(* Logix 5000 project; controller STAT 1756-L72 rev 20.12; software revision 20.04; part 28 of 34 *)
(* tags used below, declared in another part *)
   B3 : DINT[35];
   N20 : DINT[50];
   N7 : DINT[150];
   N9 : DINT[200];
   T4 : TIMER[100];
   L2_L3_ppas : DINT;
   l2va2 : BOOL;
   l2va3 : BOOL;
   l3va1 : BOOL;
   l3va2 : BOOL;
   l3va3 : BOOL;
   l3va4 : BOOL;
   naohL1VA4 : BOOL;
   naohL2VA4 : BOOL;
   stocklancy3 : DINT;
(* LANCY, continued *)

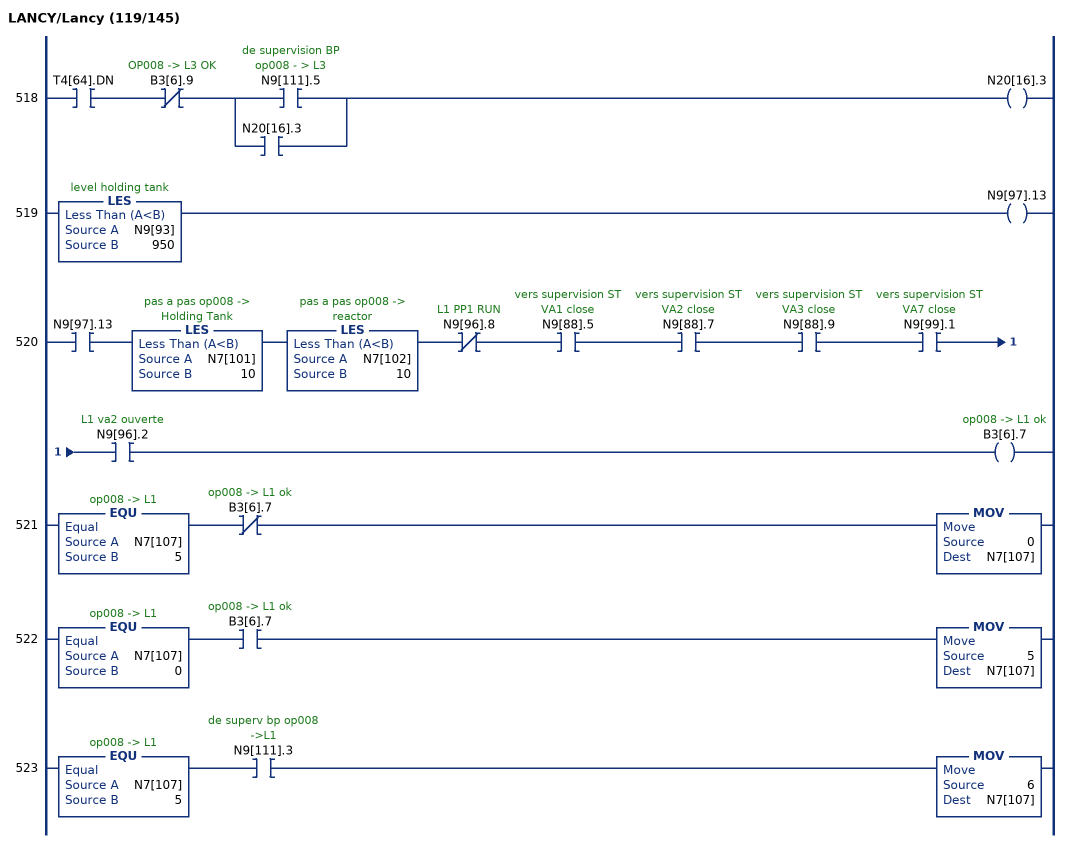
   518: XIC(T4[64].DN)XIO(B3[6].9)[XIC(N9[111].5) ,XIC(N20[16].3) ]OTE(N20[16].3);
   519: LES(N9[93],950)OTE(N9[97].13);
   520: XIC(N9[97].13)LES(N7[101],10)LES(N7[102],10)XIO(N9[96].8)XIC(N9[88].5)XIC(N9[88].7)XIC(N9[88].9)XIC(N9[99].1)XIC(N9[96].2)OTE(B3[6].7);
   521: EQU(N7[107],5)XIO(B3[6].7)MOV(0,N7[107]);
   522: EQU(N7[107],0)XIC(B3[6].7)MOV(5,N7[107]);
   523: EQU(N7[107],5)XIC(N9[111].3)MOV(6,N7[107]);
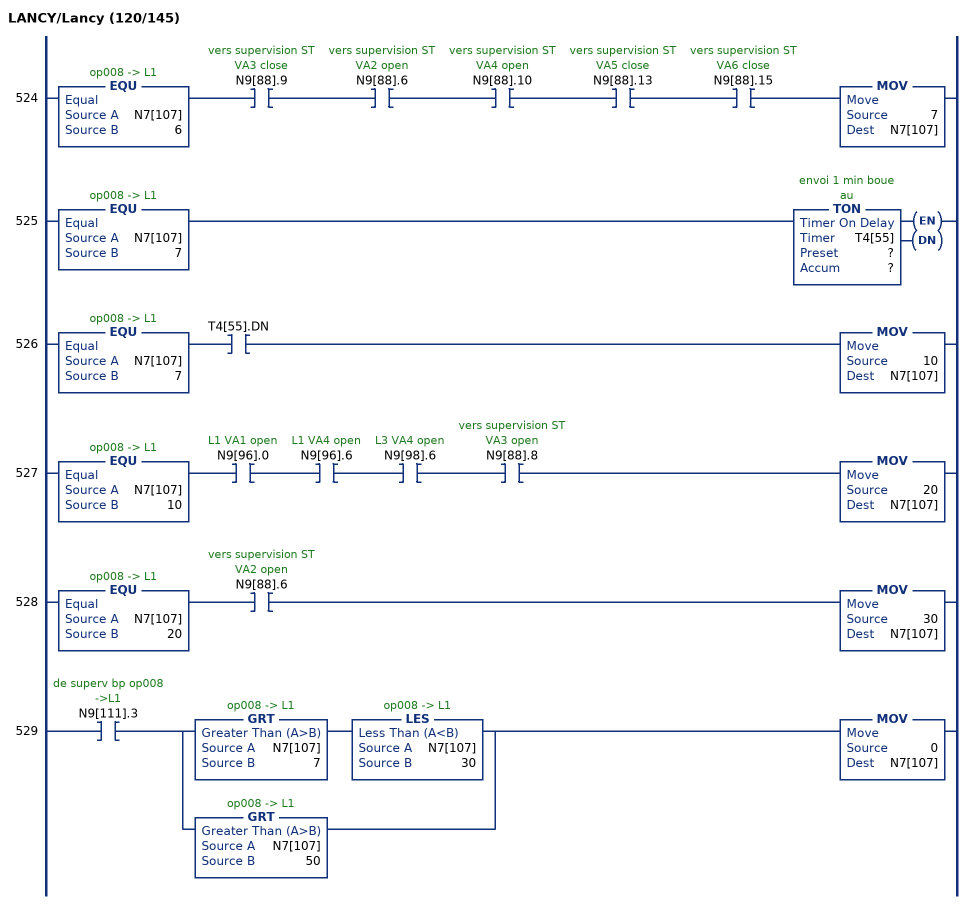
   524: EQU(N7[107],6)XIC(N9[88].9)XIC(N9[88].6)XIC(N9[88].10)XIC(N9[88].13)XIC(N9[88].15)MOV(7,N7[107]);
   525: EQU(N7[107],7)TON(T4[55],?,?);
   526: EQU(N7[107],7)XIC(T4[55].DN)MOV(10,N7[107]);
   527: EQU(N7[107],10)XIC(N9[96].0)XIC(N9[96].6)XIC(N9[98].6)XIC(N9[88].8)MOV(20,N7[107]);
   528: EQU(N7[107],20)XIC(N9[88].6)MOV(30,N7[107]);
   529: XIC(N9[111].3)[GRT(N7[107],7) LES(N7[107],30) ,GRT(N7[107],50) ]MOV(0,N7[107]);
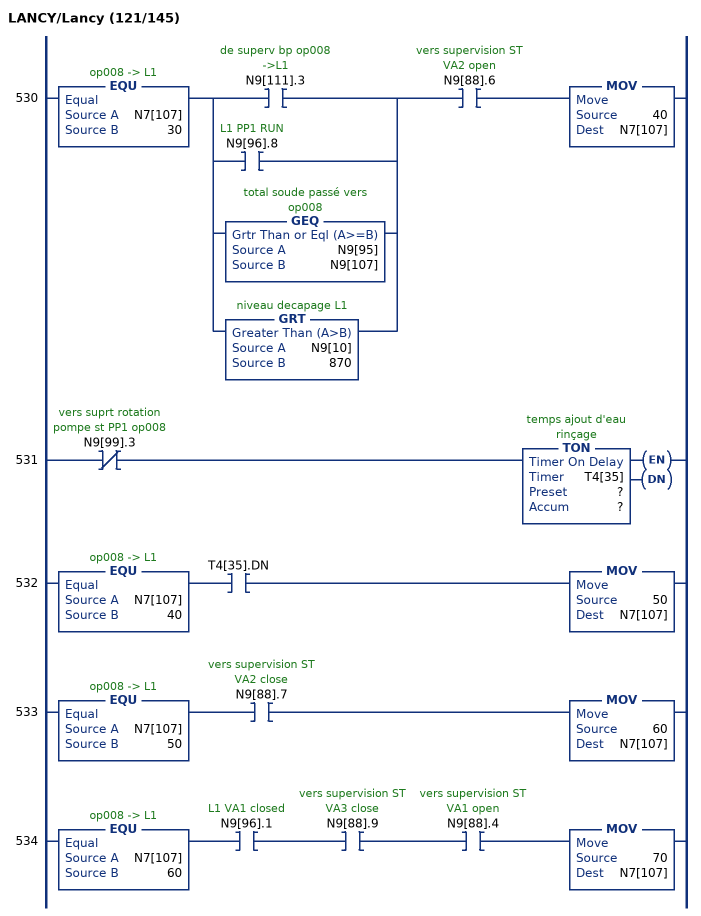
   530: EQU(N7[107],30)[XIC(N9[111].3) ,XIC(N9[96].8) ,GEQ(N9[95],N9[107]) ,GRT(N9[10],870) ]XIC(N9[88].6)MOV(40,N7[107]);
   531: XIO(N9[99].3)TON(T4[35],?,?);
   532: EQU(N7[107],40)XIC(T4[35].DN)MOV(50,N7[107]);
   533: EQU(N7[107],50)XIC(N9[88].7)MOV(60,N7[107]);
   534: EQU(N7[107],60)XIC(N9[96].1)XIC(N9[88].9)XIC(N9[88].4)MOV(70,N7[107]);
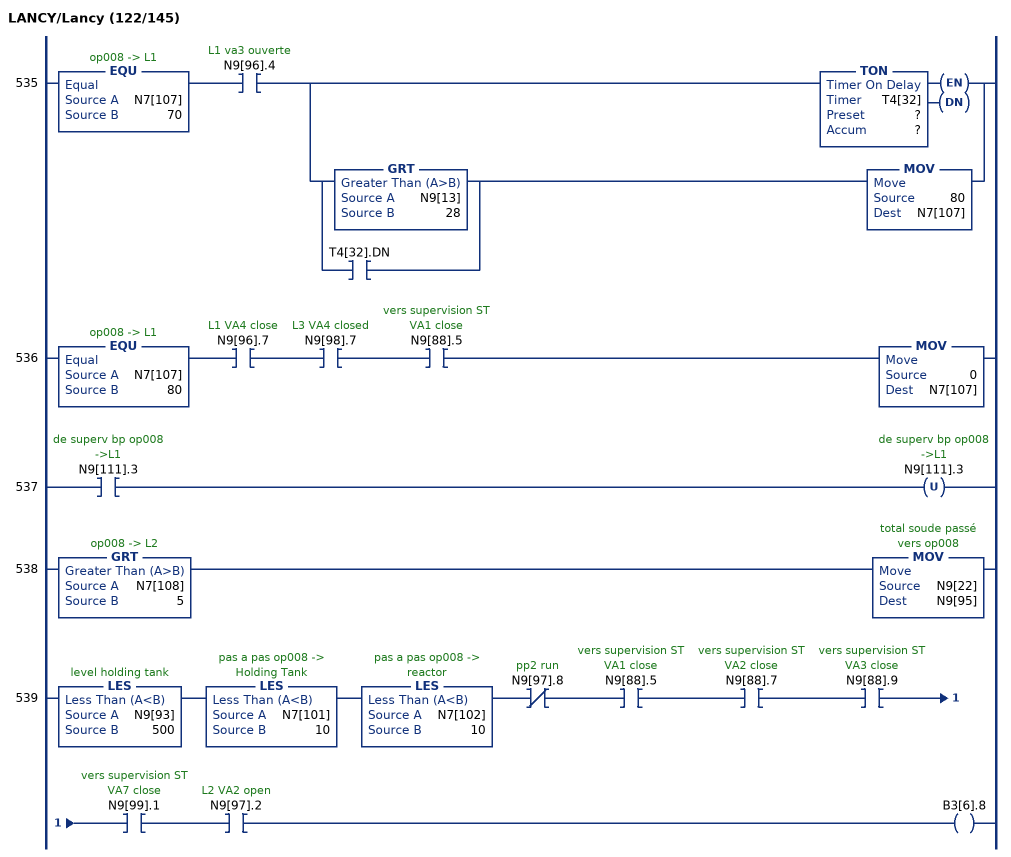
   535: EQU(N7[107],70)XIC(N9[96].4)[TON(T4[32],?,?) ,[GRT(N9[13],28) ,XIC(T4[32].DN) ] MOV(80,N7[107]) ];
   536: EQU(N7[107],80)XIC(N9[96].7)XIC(N9[98].7)XIC(N9[88].5)MOV(0,N7[107]);
   537: XIC(N9[111].3)OTU(N9[111].3);
   538: GRT(N7[108],5)MOV(N9[22],N9[95]);
   539: LES(N9[93],500)LES(N7[101],10)LES(N7[102],10)XIO(N9[97].8)XIC(N9[88].5)XIC(N9[88].7)XIC(N9[88].9)XIC(N9[99].1)XIC(N9[97].2)OTE(B3[6].8);
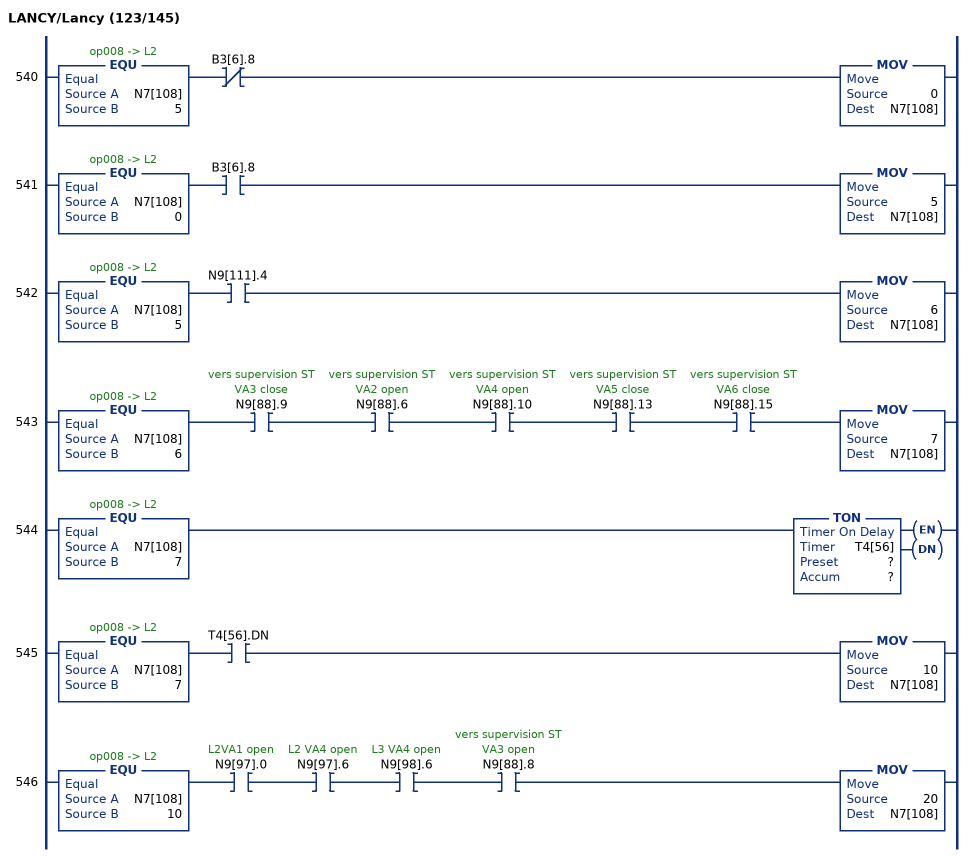
   540: EQU(N7[108],5)XIO(B3[6].8)MOV(0,N7[108]);
   541: EQU(N7[108],0)XIC(B3[6].8)MOV(5,N7[108]);
   542: EQU(N7[108],5)XIC(N9[111].4)MOV(6,N7[108]);
   543: EQU(N7[108],6)XIC(N9[88].9)XIC(N9[88].6)XIC(N9[88].10)XIC(N9[88].13)XIC(N9[88].15)MOV(7,N7[108]);
   544: EQU(N7[108],7)TON(T4[56],?,?);
   545: EQU(N7[108],7)XIC(T4[56].DN)MOV(10,N7[108]);
   546: EQU(N7[108],10)XIC(N9[97].0)XIC(N9[97].6)XIC(N9[98].6)XIC(N9[88].8)MOV(20,N7[108]);
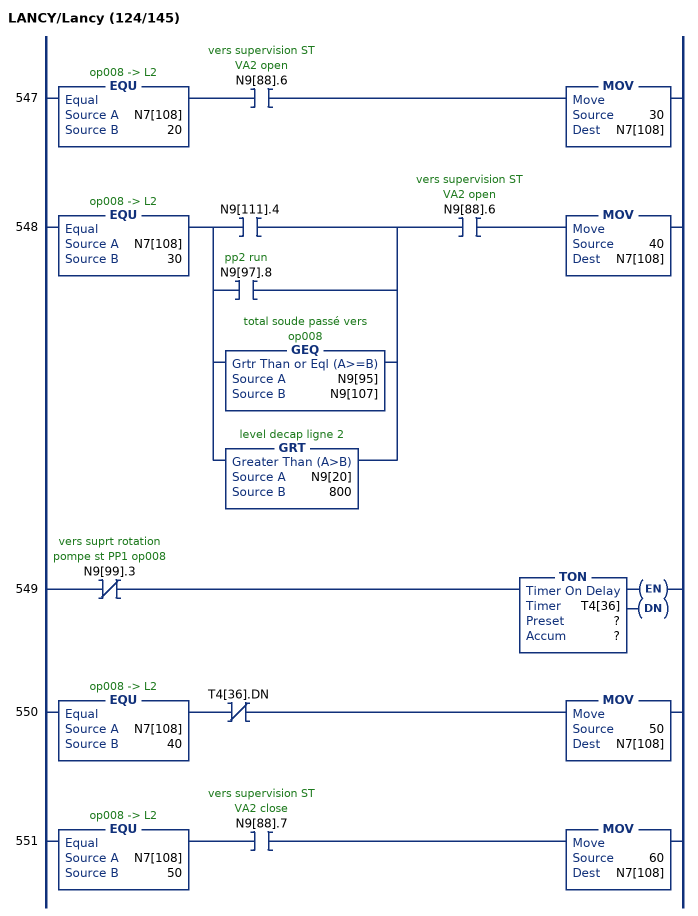
   547: EQU(N7[108],20)XIC(N9[88].6)MOV(30,N7[108]);
   548: EQU(N7[108],30)[XIC(N9[111].4) ,XIC(N9[97].8) ,GEQ(N9[95],N9[107]) ,GRT(N9[20],800) ]XIC(N9[88].6)MOV(40,N7[108]);
   549: XIO(N9[99].3)TON(T4[36],?,?);
   550: EQU(N7[108],40)XIO(T4[36].DN)MOV(50,N7[108]);
   551: EQU(N7[108],50)XIC(N9[88].7)MOV(60,N7[108]);
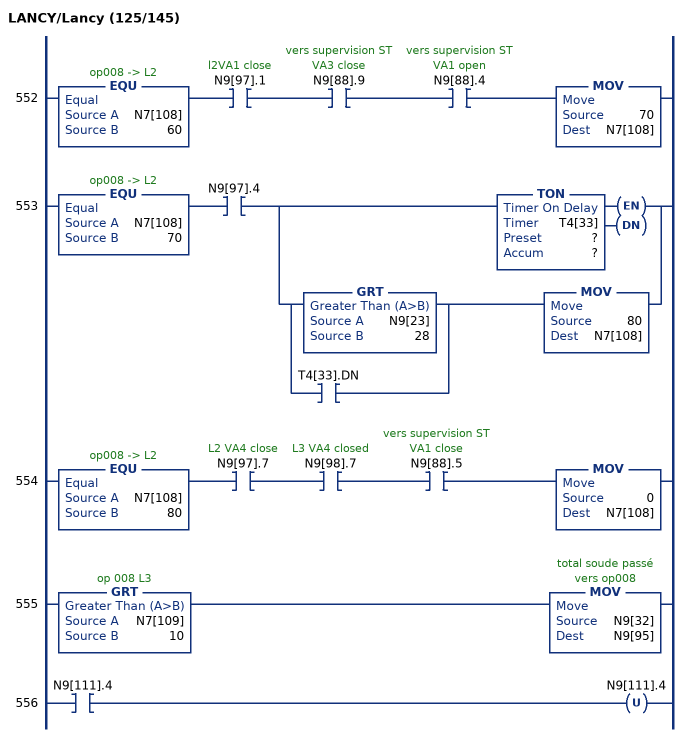
   552: EQU(N7[108],60)XIC(N9[97].1)XIC(N9[88].9)XIC(N9[88].4)MOV(70,N7[108]);
   553: EQU(N7[108],70)XIC(N9[97].4)[TON(T4[33],?,?) ,[GRT(N9[23],28) ,XIC(T4[33].DN) ] MOV(80,N7[108]) ];
   554: EQU(N7[108],80)XIC(N9[97].7)XIC(N9[98].7)XIC(N9[88].5)MOV(0,N7[108]);
   555: GRT(N7[109],10)MOV(N9[32],N9[95]);
   556: XIC(N9[111].4)OTU(N9[111].4);
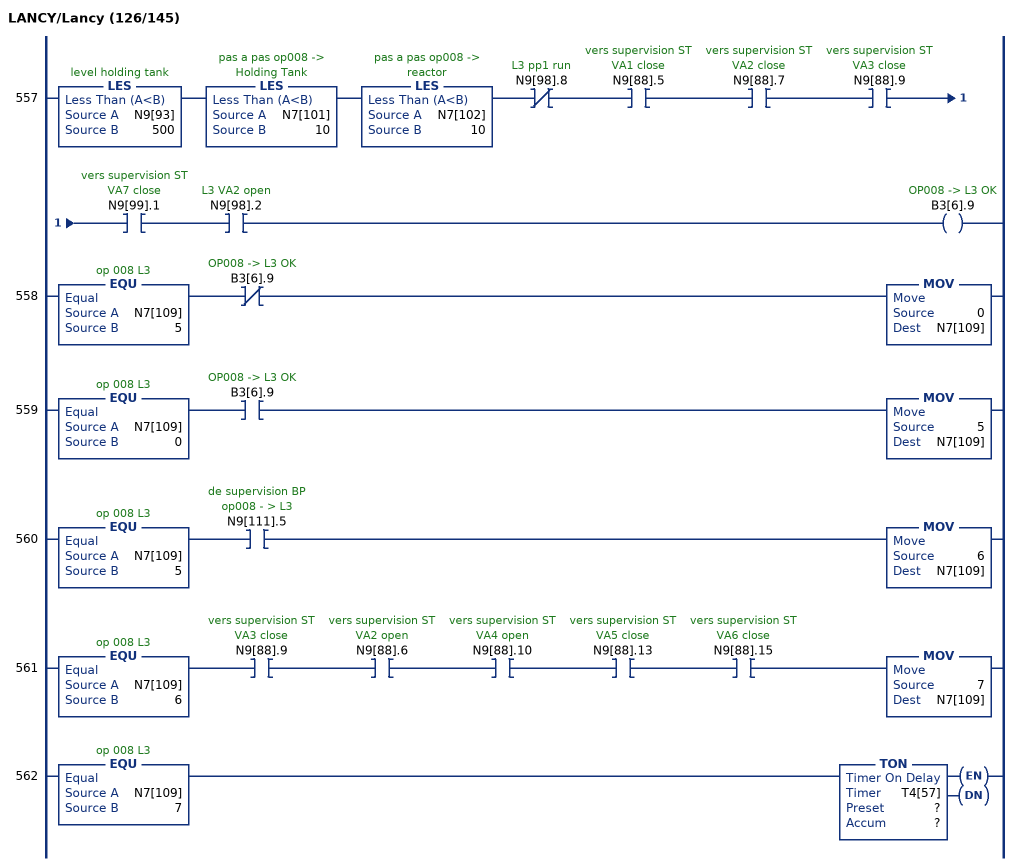
   557: LES(N9[93],500)LES(N7[101],10)LES(N7[102],10)XIO(N9[98].8)XIC(N9[88].5)XIC(N9[88].7)XIC(N9[88].9)XIC(N9[99].1)XIC(N9[98].2)OTE(B3[6].9);
   558: EQU(N7[109],5)XIO(B3[6].9)MOV(0,N7[109]);
   559: EQU(N7[109],0)XIC(B3[6].9)MOV(5,N7[109]);
   560: EQU(N7[109],5)XIC(N9[111].5)MOV(6,N7[109]);
   561: EQU(N7[109],6)XIC(N9[88].9)XIC(N9[88].6)XIC(N9[88].10)XIC(N9[88].13)XIC(N9[88].15)MOV(7,N7[109]);
   562: EQU(N7[109],7)TON(T4[57],?,?);
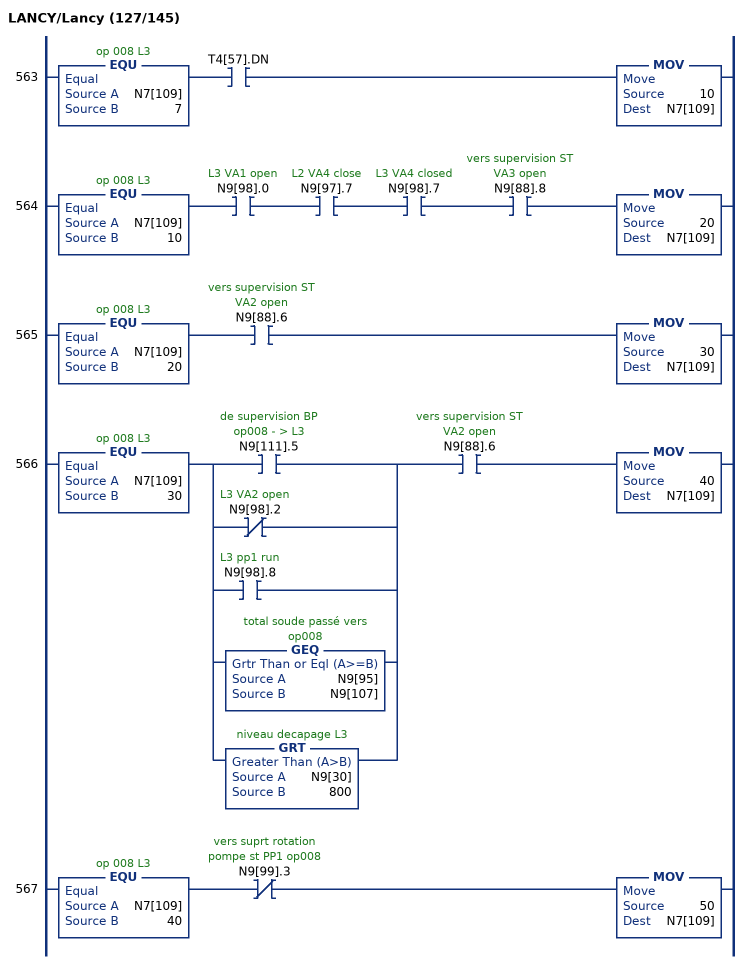
   563: EQU(N7[109],7)XIC(T4[57].DN)MOV(10,N7[109]);
   564: EQU(N7[109],10)XIC(N9[98].0)XIC(N9[97].7)XIC(N9[98].7)XIC(N9[88].8)MOV(20,N7[109]);
   565: EQU(N7[109],20)XIC(N9[88].6)MOV(30,N7[109]);
   566: EQU(N7[109],30)[XIC(N9[111].5) ,XIO(N9[98].2) ,XIC(N9[98].8) ,GEQ(N9[95],N9[107]) ,GRT(N9[30],800) ]XIC(N9[88].6)MOV(40,N7[109]);
   567: EQU(N7[109],40)XIO(N9[99].3)MOV(50,N7[109]);
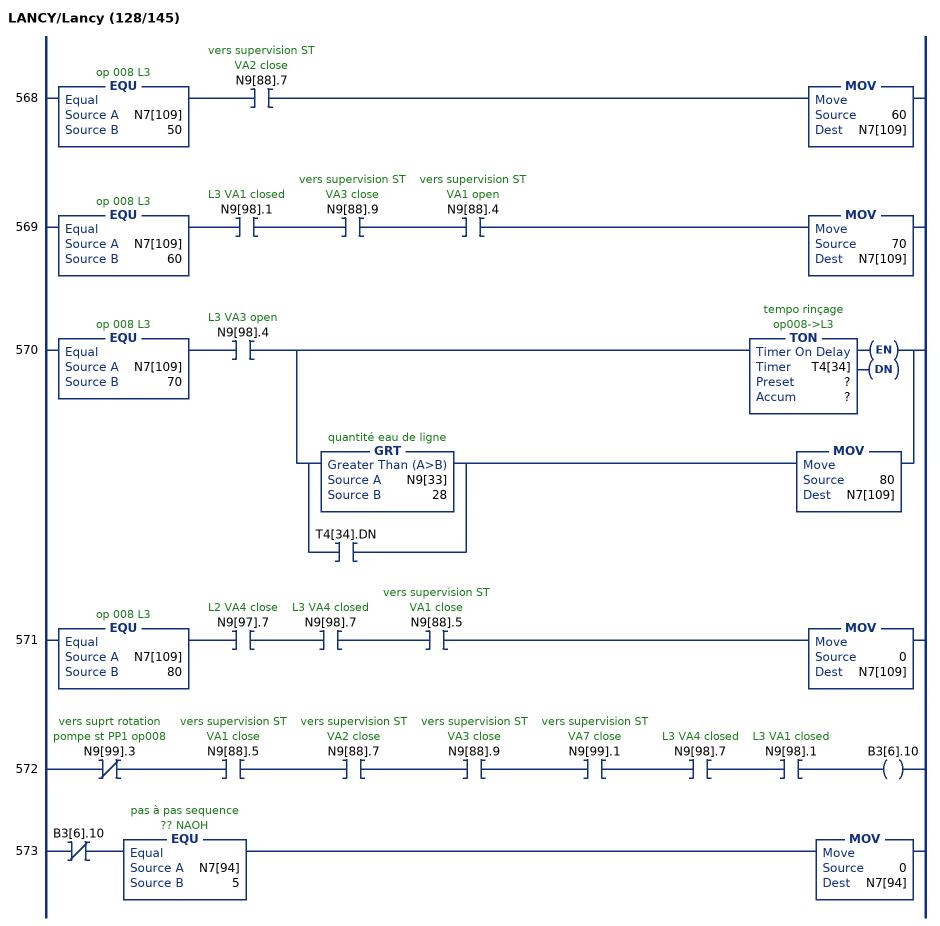
   568: EQU(N7[109],50)XIC(N9[88].7)MOV(60,N7[109]);
   569: EQU(N7[109],60)XIC(N9[98].1)XIC(N9[88].9)XIC(N9[88].4)MOV(70,N7[109]);
   570: EQU(N7[109],70)XIC(N9[98].4)[TON(T4[34],?,?) ,[GRT(N9[33],28) ,XIC(T4[34].DN) ] MOV(80,N7[109]) ];
   571: EQU(N7[109],80)XIC(N9[97].7)XIC(N9[98].7)XIC(N9[88].5)MOV(0,N7[109]);
   572: XIO(N9[99].3)XIC(N9[88].5)XIC(N9[88].7)XIC(N9[88].9)XIC(N9[99].1)XIC(N9[98].7)XIC(N9[98].1)OTE(B3[6].10);
   573: XIO(B3[6].10)EQU(N7[94],5)MOV(0,N7[94]);
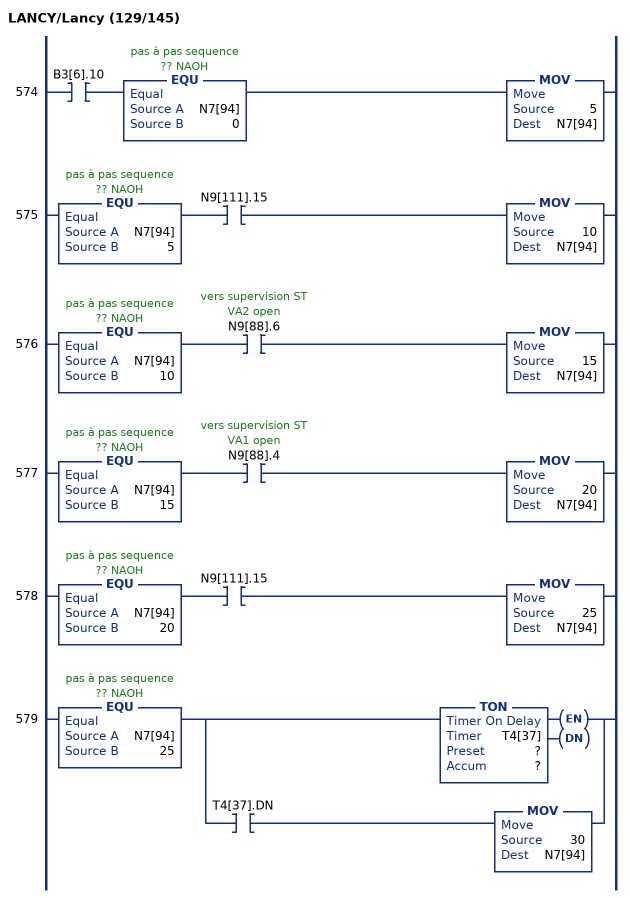
   574: XIC(B3[6].10)EQU(N7[94],0)MOV(5,N7[94]);
   575: EQU(N7[94],5)XIC(N9[111].15)MOV(10,N7[94]);
   576: EQU(N7[94],10)XIC(N9[88].6)MOV(15,N7[94]);
   577: EQU(N7[94],15)XIC(N9[88].4)MOV(20,N7[94]);
   578: EQU(N7[94],20)XIC(N9[111].15)MOV(25,N7[94]);
   579: EQU(N7[94],25)[TON(T4[37],?,?) ,XIC(T4[37].DN) MOV(30,N7[94]) ];
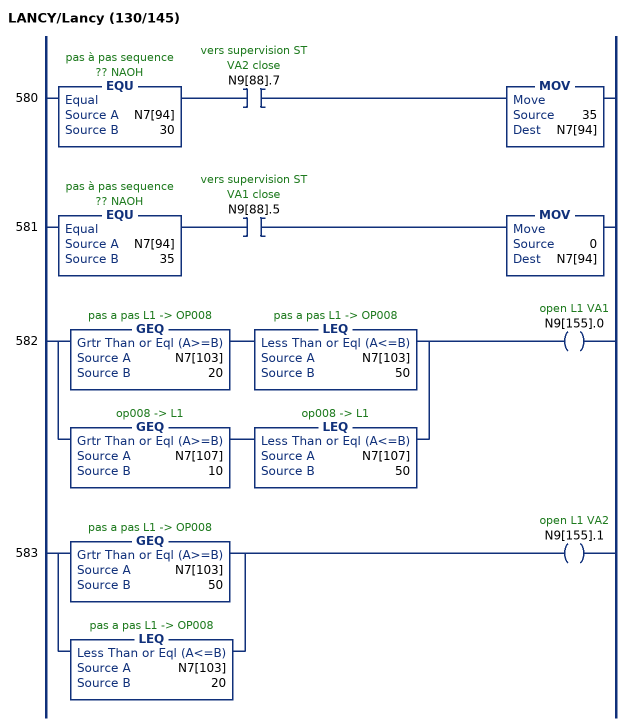
   580: EQU(N7[94],30)XIC(N9[88].7)MOV(35,N7[94]);
   581: EQU(N7[94],35)XIC(N9[88].5)MOV(0,N7[94]);
   582: [GEQ(N7[103],20) LEQ(N7[103],50) ,GEQ(N7[107],10) LEQ(N7[107],50) ]OTE(N9[155].0);
   583: [GEQ(N7[103],50) ,LEQ(N7[103],20) ]OTE(N9[155].1);
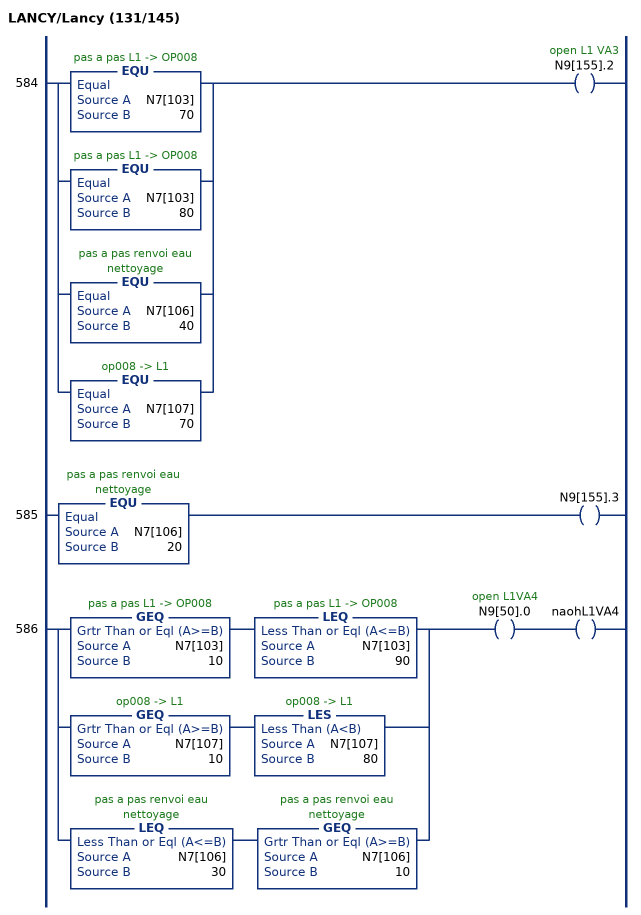
   584: [EQU(N7[103],70) ,EQU(N7[103],80) ,EQU(N7[106],40) ,EQU(N7[107],70) ]OTE(N9[155].2);
   585: EQU(N7[106],20)OTE(N9[155].3);
   586: [GEQ(N7[103],10) LEQ(N7[103],90) ,GEQ(N7[107],10) LES(N7[107],80) ,LEQ(N7[106],30) GEQ(N7[106],10) ]OTE(N9[50].0)OTE(naohL1VA4);
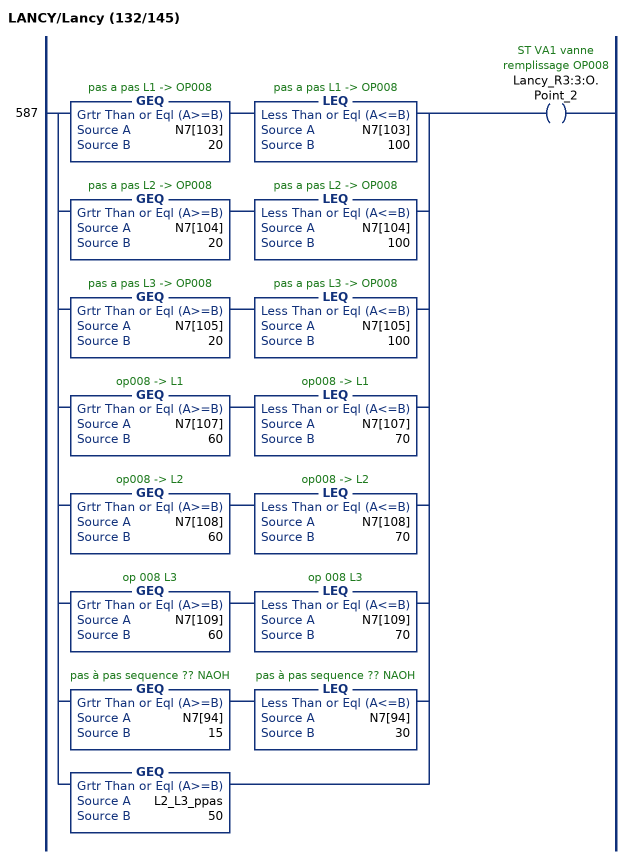
   587: [GEQ(N7[103],20) LEQ(N7[103],100) ,GEQ(N7[104],20) LEQ(N7[104],100) ,GEQ(N7[105],20) LEQ(N7[105],100) ,GEQ(N7[107],60) LEQ(N7[107],70) ,GEQ(N7[108],60) LEQ(N7[108],70) ,GEQ(N7[109],60) LEQ(N7[109],70) ,GEQ(N7[94],15) LEQ(N7[94],30) ,GEQ(L2_L3_ppas,50) ]OTE(Lancy_R3:3:O.Point_2);
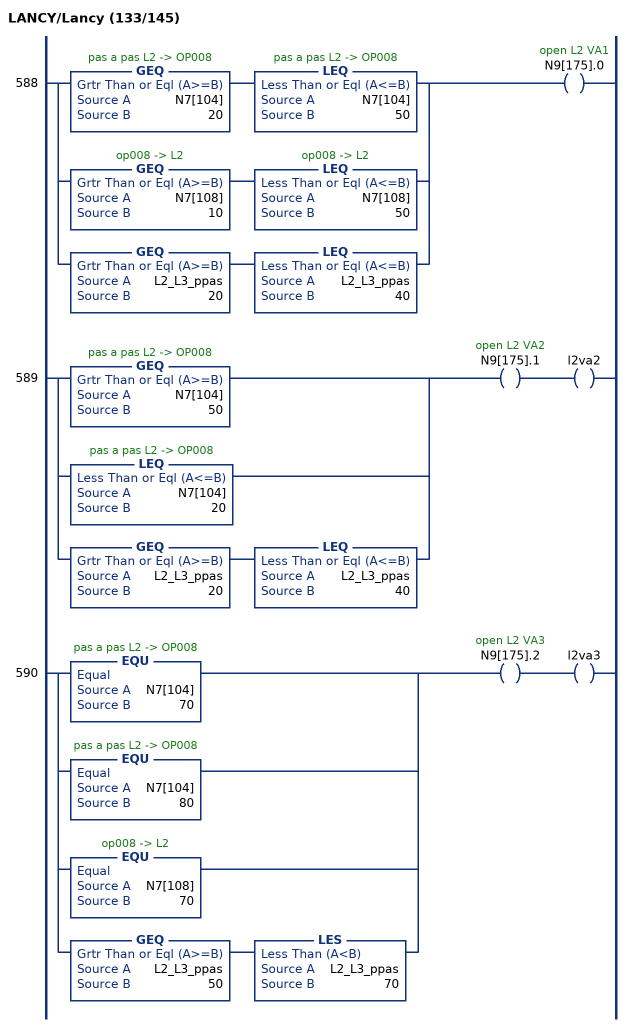
   588: [GEQ(N7[104],20) LEQ(N7[104],50) ,GEQ(N7[108],10) LEQ(N7[108],50) ,GEQ(L2_L3_ppas,20) LEQ(L2_L3_ppas,40) ]OTE(N9[175].0);
   589: [GEQ(N7[104],50) ,LEQ(N7[104],20) ,GEQ(L2_L3_ppas,20) LEQ(L2_L3_ppas,40) ]OTE(N9[175].1)OTE(l2va2);
   590: [EQU(N7[104],70) ,EQU(N7[104],80) ,EQU(N7[108],70) ,GEQ(L2_L3_ppas,50) LES(L2_L3_ppas,70) ]OTE(N9[175].2)OTE(l2va3);
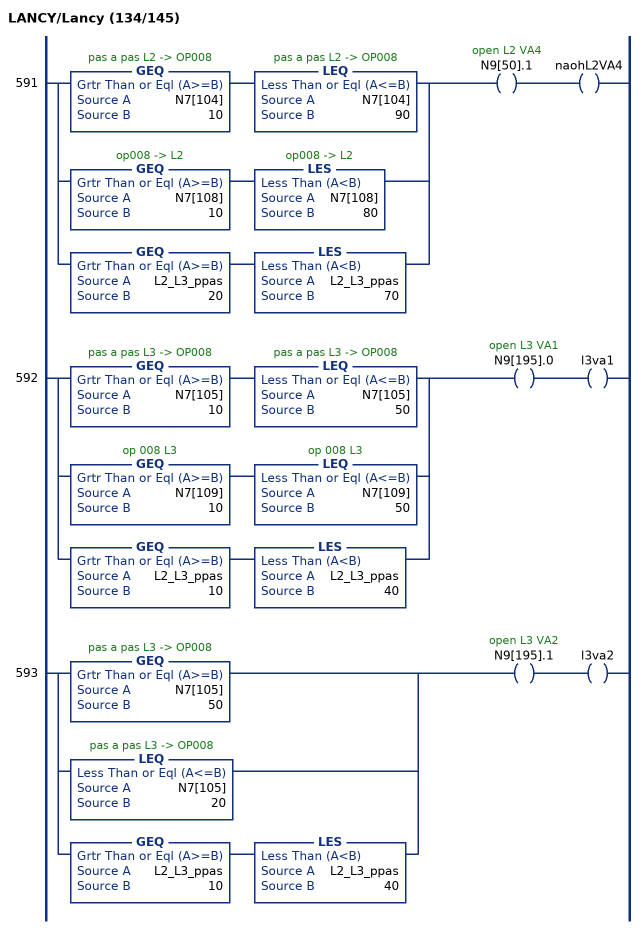
   591: [GEQ(N7[104],10) LEQ(N7[104],90) ,GEQ(N7[108],10) LES(N7[108],80) ,GEQ(L2_L3_ppas,20) LES(L2_L3_ppas,70) ]OTE(N9[50].1)OTE(naohL2VA4);
   592: [GEQ(N7[105],10) LEQ(N7[105],50) ,GEQ(N7[109],10) LEQ(N7[109],50) ,GEQ(L2_L3_ppas,10) LES(L2_L3_ppas,40) ]OTE(N9[195].0)OTE(l3va1);
   593: [GEQ(N7[105],50) ,LEQ(N7[105],20) ,GEQ(L2_L3_ppas,10) LES(L2_L3_ppas,40) ]OTE(N9[195].1)OTE(l3va2);
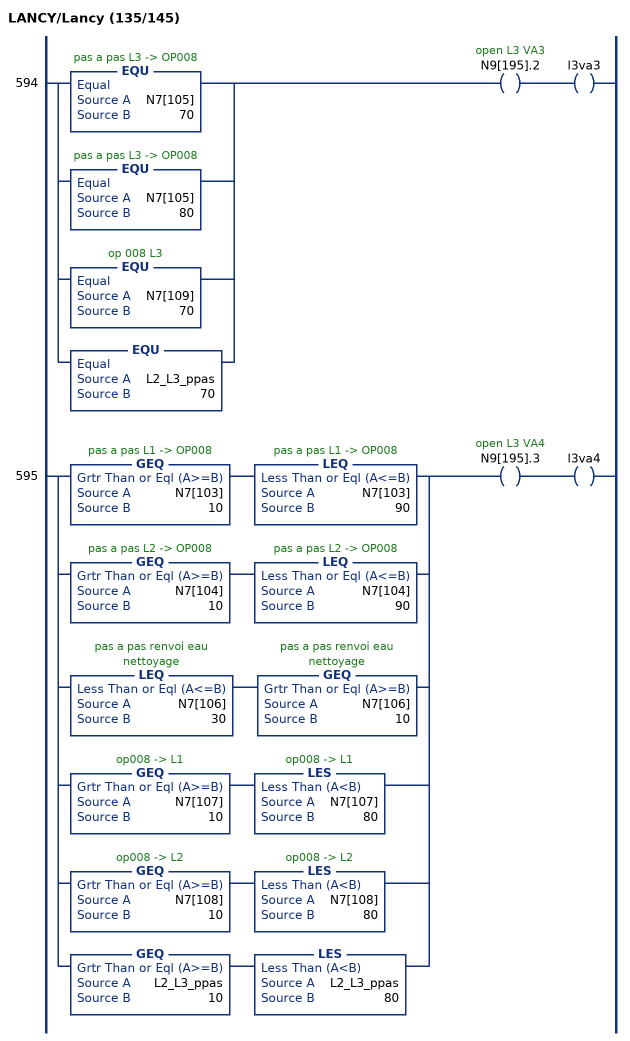
   594: [EQU(N7[105],70) ,EQU(N7[105],80) ,EQU(N7[109],70) ,EQU(L2_L3_ppas,70) ]OTE(N9[195].2)OTE(l3va3);
   595: [GEQ(N7[103],10) LEQ(N7[103],90) ,GEQ(N7[104],10) LEQ(N7[104],90) ,LEQ(N7[106],30) GEQ(N7[106],10) ,GEQ(N7[107],10) LES(N7[107],80) ,GEQ(N7[108],10) LES(N7[108],80) ,GEQ(L2_L3_ppas,10) LES(L2_L3_ppas,80) ]OTE(N9[195].3)OTE(l3va4);
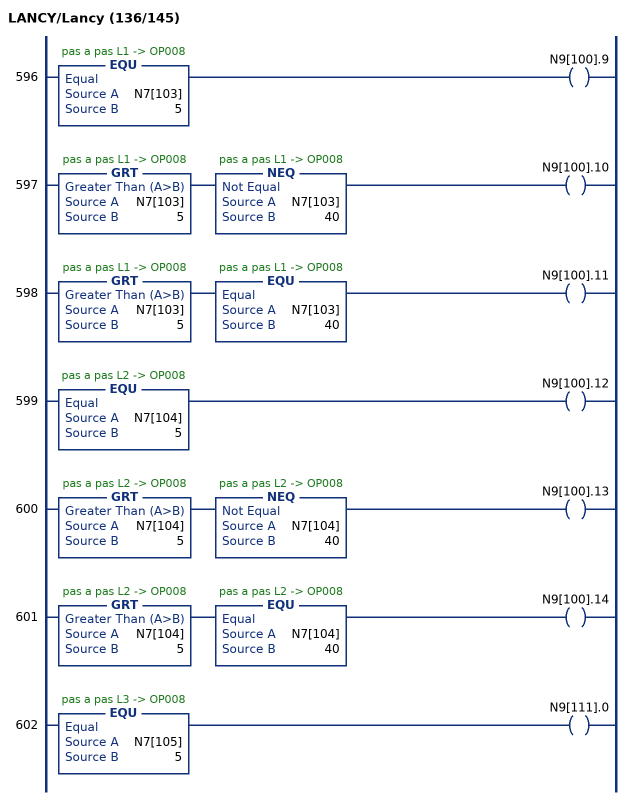
   596: EQU(N7[103],5)OTE(N9[100].9);
   597: GRT(N7[103],5)NEQ(N7[103],40)OTE(N9[100].10);
   598: GRT(N7[103],5)EQU(N7[103],40)OTE(N9[100].11);
   599: EQU(N7[104],5)OTE(N9[100].12);
   600: GRT(N7[104],5)NEQ(N7[104],40)OTE(N9[100].13);
   601: GRT(N7[104],5)EQU(N7[104],40)OTE(N9[100].14);
   602: EQU(N7[105],5)OTE(N9[111].0);
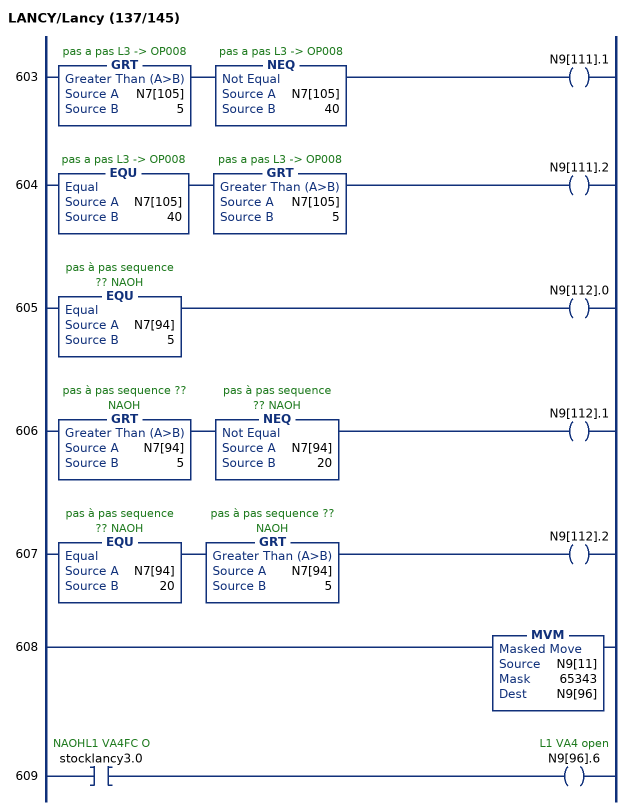
   603: GRT(N7[105],5)NEQ(N7[105],40)OTE(N9[111].1);
   604: EQU(N7[105],40)GRT(N7[105],5)OTE(N9[111].2);
   605: EQU(N7[94],5)OTE(N9[112].0);
   606: GRT(N7[94],5)NEQ(N7[94],20)OTE(N9[112].1);
   607: EQU(N7[94],20)GRT(N7[94],5)OTE(N9[112].2);
   608: MVM(N9[11],65343,N9[96]);
   609: XIC(stocklancy3.0)OTE(N9[96].6);
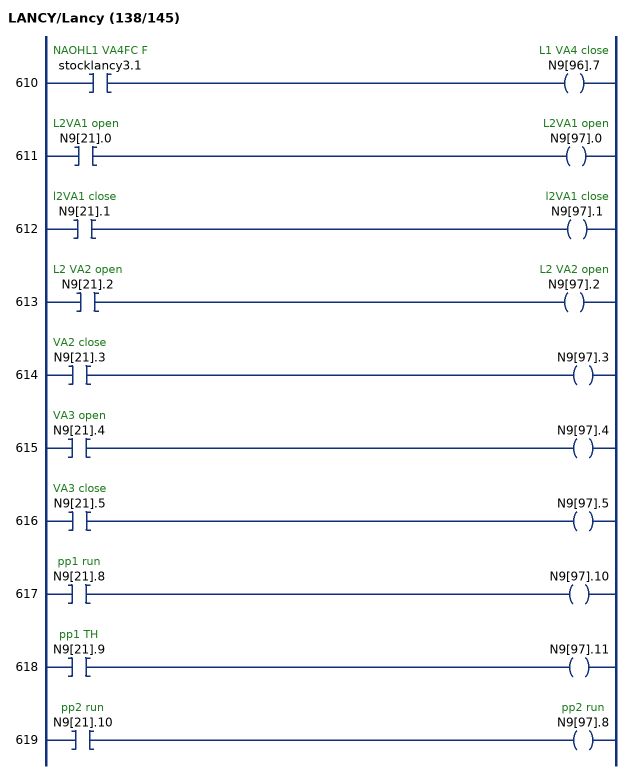
   610: XIC(stocklancy3.1)OTE(N9[96].7);
   611: XIC(N9[21].0)OTE(N9[97].0);
   612: XIC(N9[21].1)OTE(N9[97].1);
   613: XIC(N9[21].2)OTE(N9[97].2);
   614: XIC(N9[21].3)OTE(N9[97].3);
   615: XIC(N9[21].4)OTE(N9[97].4);
   616: XIC(N9[21].5)OTE(N9[97].5);
   617: XIC(N9[21].8)OTE(N9[97].10);
   618: XIC(N9[21].9)OTE(N9[97].11);
   619: XIC(N9[21].10)OTE(N9[97].8);
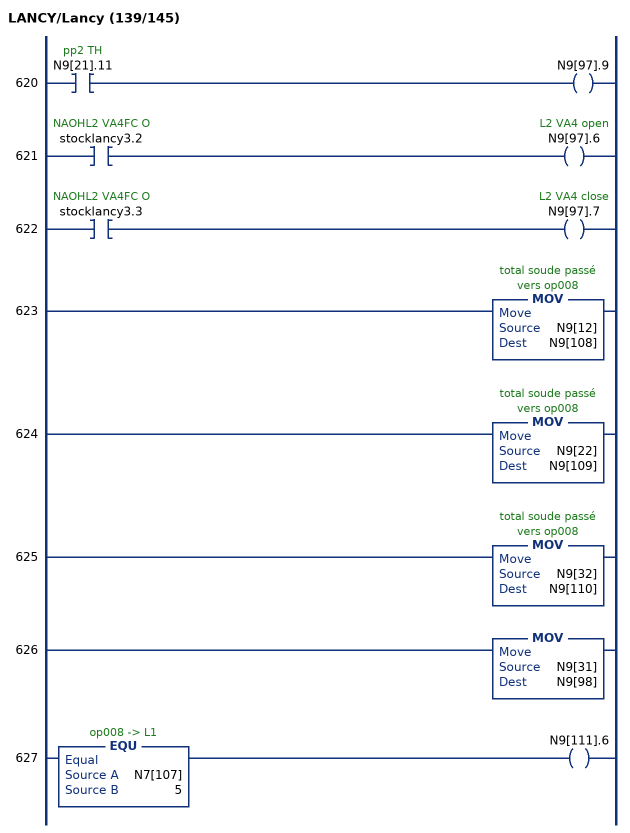
   620: XIC(N9[21].11)OTE(N9[97].9);
   621: XIC(stocklancy3.2)OTE(N9[97].6);
   622: XIC(stocklancy3.3)OTE(N9[97].7);
   623: MOV(N9[12],N9[108]);
   624: MOV(N9[22],N9[109]);
   625: MOV(N9[32],N9[110]);
   626: MOV(N9[31],N9[98]);
   627: EQU(N7[107],5)OTE(N9[111].6);
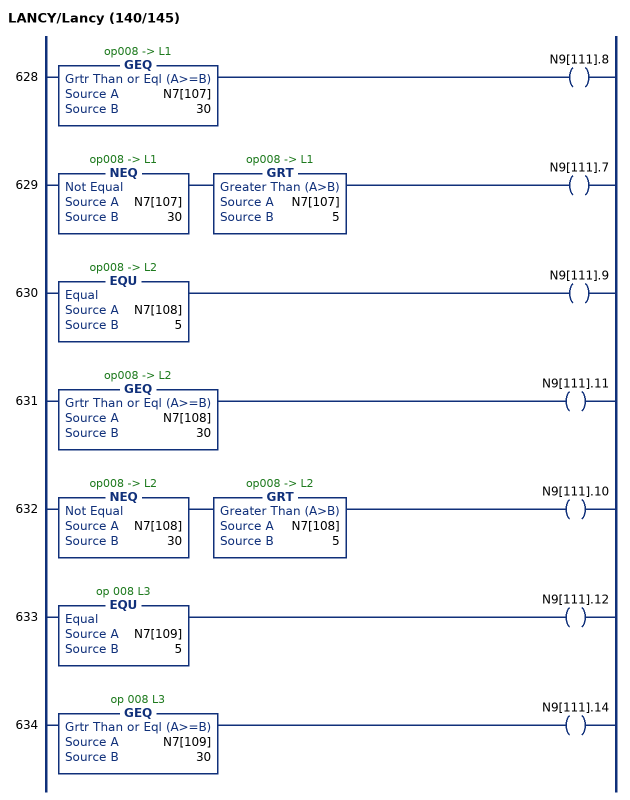
   628: GEQ(N7[107],30)OTE(N9[111].8);
   629: NEQ(N7[107],30)GRT(N7[107],5)OTE(N9[111].7);
   630: EQU(N7[108],5)OTE(N9[111].9);
   631: GEQ(N7[108],30)OTE(N9[111].11);
   632: NEQ(N7[108],30)GRT(N7[108],5)OTE(N9[111].10);
   633: EQU(N7[109],5)OTE(N9[111].12);
   634: GEQ(N7[109],30)OTE(N9[111].14);
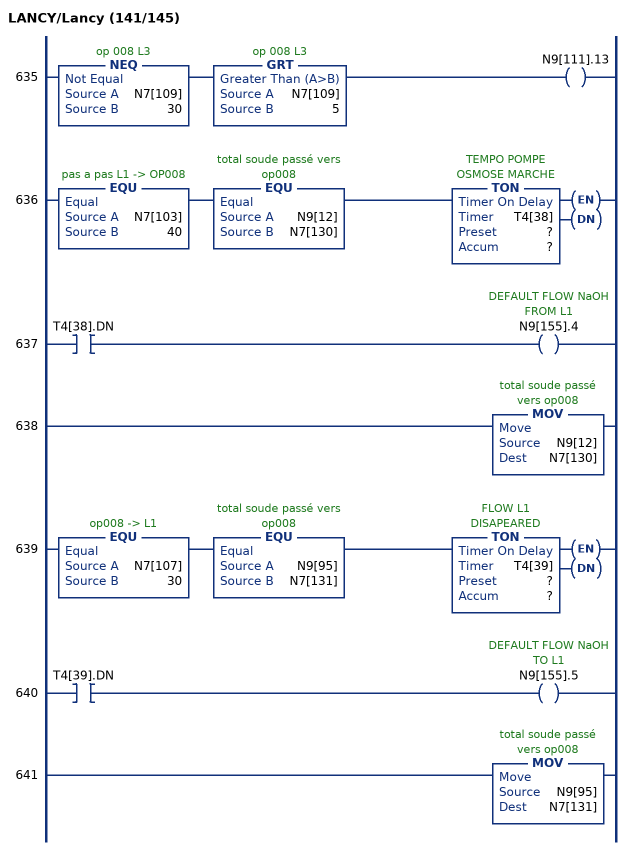
   635: NEQ(N7[109],30)GRT(N7[109],5)OTE(N9[111].13);
   636: EQU(N7[103],40)EQU(N9[12],N7[130])TON(T4[38],?,?);
   637: XIC(T4[38].DN)OTE(N9[155].4);
   638: MOV(N9[12],N7[130]);
   639: EQU(N7[107],30)EQU(N9[95],N7[131])TON(T4[39],?,?);
   640: XIC(T4[39].DN)OTE(N9[155].5);
   641: MOV(N9[95],N7[131]);
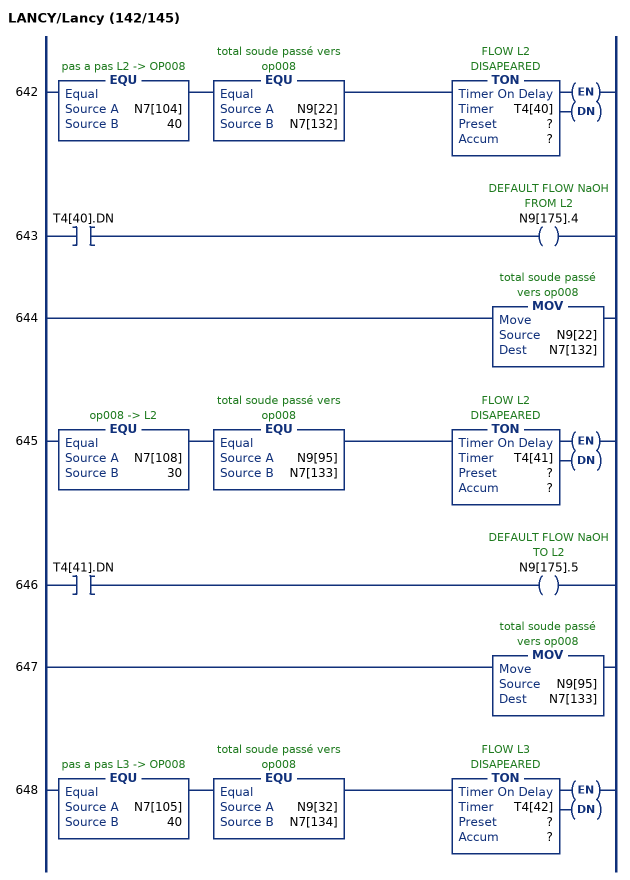
   642: EQU(N7[104],40)EQU(N9[22],N7[132])TON(T4[40],?,?);
   643: XIC(T4[40].DN)OTE(N9[175].4);
   644: MOV(N9[22],N7[132]);
   645: EQU(N7[108],30)EQU(N9[95],N7[133])TON(T4[41],?,?);
   646: XIC(T4[41].DN)OTE(N9[175].5);
   647: MOV(N9[95],N7[133]);
   648: EQU(N7[105],40)EQU(N9[32],N7[134])TON(T4[42],?,?);
